// TIA Portal V17 export
// export: Created 2025-03-07T09:23:55.2966294Z, ExportSetting WithDefaults, DisplayName Totally Integrated Automation Portal, DisplayVersion V17 Update 8, DisplayName TIA Portal Openness, DisplayVersion V17 Update 8, DisplayName TIA Portal Version Control Interface, DisplayVersion V17, DisplayName SINAMICS Startdrive Advanced, DisplayVersion V17 SP2, DisplayName SINAMICS Startdrive G110M, G120, G120C, G120D, G120P, G115D, DisplayVersion V17 SP2, DisplayName SINAMICS Startdrive G130, G150, S120, S150, SINAMICS MV, S210, DisplayVersion V17 SP2, DisplayName STEP 7 Professional, DisplayVersion V17 Update 8, DisplayName SINUMERIK ONE STEP 7 Toolbox, DisplayVersion V17 Update 12, DisplayName SINUMERIK 840D sl STEP 7 Toolbox, DisplayVersion V17 Update 12, DisplayName STEP 7 Safety, DisplayVersion V17 Update 6, DisplayName WinCC Advanced, DisplayVersion V17 Update 8
FUNCTION "FC21020_FEEDER_SCALING" : Void   // FC21020, LAD
TITLE = Robot-PLC Scaling
{ S7_Optimized_Access := 'TRUE' }
AUTHOR : Jbarturen
VERSION : 0.1
// stored: AutoNumber false, IsIECCheckEnabled false, SetENOAutomatically false, UDAEnableTagReadback false
   VAR_INPUT
      DINT_INPUT_VALUE : DInt;
      REAL_INPUT_VALUE : Real;
      DINT_TO_REAL : Bool;
      REAL_TRANSFORM_FOR_FEEDER : Bool;
   END_VAR
   VAR_OUTPUT
      OUTPUT_VALUE_PLC : Real;
      OUTPUT_VALUE_FEEDER : Real;
   END_VAR
   VAR_TEMP
      Value_Swapped : DInt;
      Value_Real : Real;
      Value_PLC : Real;
      Value_DWord : DWord;
      Value_DWord_Swapped : DWord;
   END_VAR
BEGIN

REGION Network 1: DATA TYPE CONVERTION / Robot-PLC
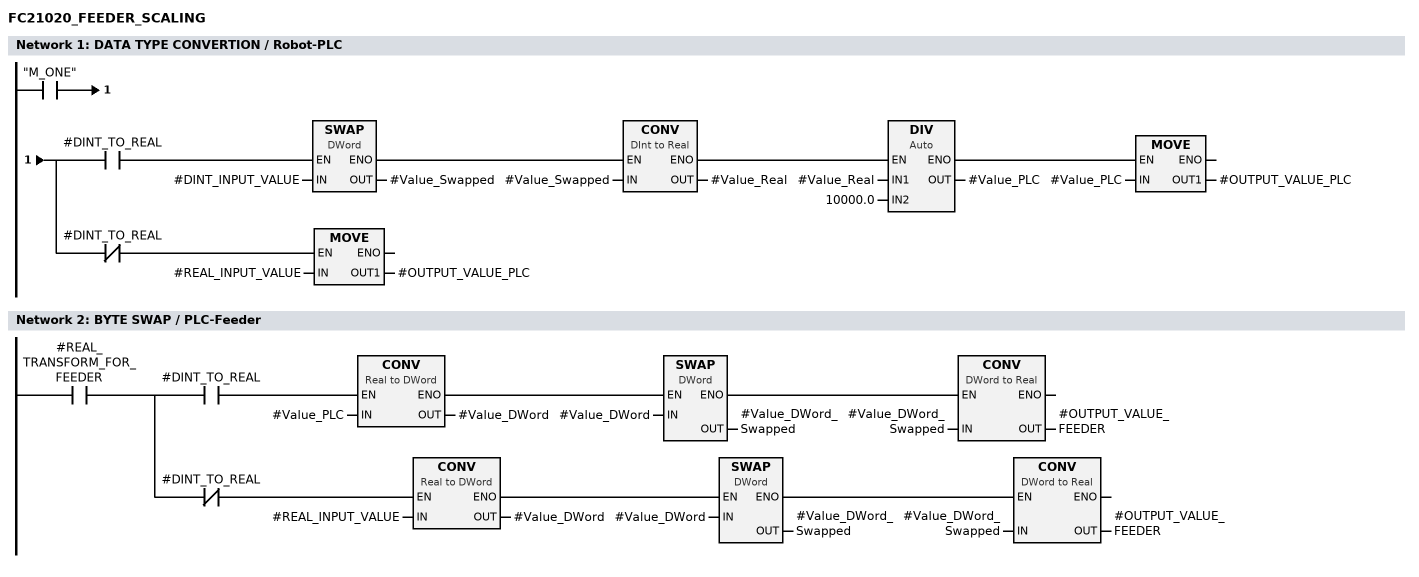
   IF "M_ONE" AND #DINT_TO_REAL THEN
       #Value_Swapped := SWAP(#DINT_INPUT_VALUE);
       #Value_Real := DINT_TO_REAL(#Value_Swapped);
       #Value_PLC := #Value_Real / 10000.0;
       #OUTPUT_VALUE_PLC := #Value_PLC;
   END_IF;
   IF "M_ONE" AND NOT #DINT_TO_REAL THEN #OUTPUT_VALUE_PLC := #REAL_INPUT_VALUE; END_IF;
END_REGION

REGION Network 2: BYTE SWAP / PLC-Feeder
   IF #REAL_TRANSFORM_FOR_FEEDER AND #DINT_TO_REAL THEN
       #Value_DWord := REAL_TO_DWORD(#Value_PLC);
       #Value_DWord_Swapped := SWAP(#Value_DWord);
       #OUTPUT_VALUE_FEEDER := DWORD_TO_REAL(#Value_DWord_Swapped);
   END_IF;
   IF #REAL_TRANSFORM_FOR_FEEDER AND NOT #DINT_TO_REAL THEN
       #Value_DWord := REAL_TO_DWORD(#REAL_INPUT_VALUE);
       #Value_DWord_Swapped := SWAP(#Value_DWord);
       #OUTPUT_VALUE_FEEDER := DWORD_TO_REAL(#Value_DWord_Swapped);
   END_IF;
END_REGION
END_FUNCTION
